TYPE ST_PowerMonitor_InputField EXTENDS st_PQVoltageData:
STRUCT
	r_loadshare					: 	REAL;
	ACQuality					:	ST_PQGridQualityData;
	Powerlock					: 	ARRAY [1..2] OF st_PQVoltageData;
END_STRUCT
END_TYPE

(* stored: Version 1.1.0.1, ProductVersion 3.1.4026.18
   DUT ST_PowerMonitor_InputField: Id {9360fa12-e620-4f46-a1bd-2737abbc0f8d} *)
